TYPE ST_TopElement_HMI EXTENDS ST_BaseTopElement_HMI :
STRUCT
	
END_STRUCT
END_TYPE

(* stored: Version 1.1.0.1, ProductVersion 3.1.4024.15
   DUT ST_TopElement_HMI: Id {2be5f6d1-09e0-4dc9-9d6d-43798dc7dc48} *)
